FUNCTION_BLOCK FB_InFeedController
VAR_INPUT
END_VAR
VAR_OUTPUT
END_VAR
VAR
END_VAR

END_FUNCTION_BLOCK

(* stored: Version 1.1.0.1, ProductVersion 3.1.4024.16
   POU FB_InFeedController: Id {ff4e95ef-2fe1-4fc4-a99c-7d6bb92f39bb}, SpecialFunc None *)
